PROGRAM prg_Alarmbewaking
VAR
	Sensor1		AT		%I*		:BOOL; //Druk Te Hoog (True)
	Sensor2		AT		%I*		:BOOL; //Temperatuur Te Hoog (True)
	Sensor3		AT		%I*		:BOOL; //Laag vloeistof (True) In de oefening moet dit false zijn maar dit is gewoon verwarrend maak er dan NOT(..) van waar deze voorkomt in het programma
	DrukKnop	AT		%I*		:BOOL;
	
	Lamp1		AT		%Q*		:BOOL; //Druk Te Hoog
	Lamp2		AT		%Q*		:BOOL; //Temperatuur Te Hoog
	Lamp3		AT		%Q*		:BOOL; //Vloeistof Te Laag
	Lamp4		AT		%Q*		:BOOL; //TweeAlarmen
	Lamp5		AT		%Q*		:BOOL; //Drie Alarmen
	
	
	SetReset: SR;
END_VAR

Lamp1 := Sensor1;
Lamp2 := Sensor2;
Lamp3 := Sensor3;

Lamp4 := (NOT(Sensor1) AND Sensor2 AND Sensor3) OR
		 (Sensor1 AND NOT(Sensor2) AND Sensor3) OR
		 (Sensor1 AND Sensor2 AND NOT Sensor3);

SetReset(SET1:= Sensor1 AND Sensor2 AND Sensor3, RESET:=DrukKnop , Q1=> Lamp5);

END_PROGRAM

(* stored: Version 1.1.0.1, ProductVersion 3.1.4024.15
   POU prg_Alarmbewaking: Id {d816c7c6-aa67-463e-b00c-2a6330d8cd6a}, SpecialFunc None *)
